VAR_GLOBAL
	MoverInterface: ARRAY[1..grpcnt] OF DUT_XTS_Interface;
END_VAR

(* stored: Version 1.1.0.1, ProductVersion 3.1.0.25
   GVL CAInterface: Id {3ba2f8b4-3b2e-4366-8a28-27e677bac185} *)
